// TIA Portal V19 export
TYPE "UDT_ADIN"
   STRUCT
      "time" : Struct   // Delay setpoints
         on_set : Int := 0;   // Desired delay to set the memory switch
         off_set : Int := 0;   // Desired delay to reset the memory switch
         on_act : Int := 0;   // Counted delay to set the memory switch
         off_act : Int := 0;   // Counted delay to reset the memory switch
      END_STRUCT;
      setup : Struct   // Setup of switch
         comparison : Int := 0;   // 0 = ">", 1 = ">=", 2 = "<", 3 = "<="
         reference : Real := 0.0;   // Reference value to which the sensor is compared
         alarm : Bool := false;   // 0=alarm disabled, 1=alarm enabled
         triggerversion : Bool := false;   // 0=switch inactive for triggerring, 1=switch active for triggering
      END_STRUCT;
      faults : Struct   // Faults
         adin { S7_SetPoint := 'True'} : "UDT_ALARMACKN";   // Digital switch fault
         fpreset : Bool := false;   // Faceplate reset for individual treatment
      END_STRUCT;
      sim : Struct   // Simulation
         cmdon : Bool := false;   // simulation on command
         cmdoff : Bool := false;   // simulation off command
         simulated : Bool := false;   // 0=simulation off, 1=simulation on
         cmdforce : Bool := false;   // force switch command
         cmdunforce : Bool := false;   // unforce switch command
         forced : Bool := false;   // 0=unforced, 1=forced
      END_STRUCT;
      status : Struct   // Status
         rawinput : Real := 0.0;   // Raw input value
         processed : Bool := false;   // Status of input after comparison
         switch_active : Bool := false;   // Switch is Active after delay on
         alarm_monitor : Bool := false;   // Alarm is monitored
         fault : Bool := false;   // Fault is activated
      END_STRUCT;
      unit : WString;
   END_STRUCT;
END_TYPE
